FUNCTION F_ROUND_REAL : REAL
VAR_INPUT
  rInput 			: REAL;
  iDecimalPlaces 	: INT;
END_VAR
VAR
  rOutput 			: real;
  rLeftPart 		: REAL;
  Value				: dint;
END_VAR


rOutput := rInput * EXPT(10,iDecimalPlaces);
//rLeftPart := rOutput - TRUNC(rOutput);

//IF rLeftPart >= 0.5 THEN
//  rOutput := rOutput + 1;
//ElSIF rLeftPart <= -0.5 THEN
//  rOutput := rOutput - 1;
//ELSE
//  rOutput := rOutput;
//END_IF

Value := REAL_TO_DINT(rOutput);
rOutput := Value / EXPT(10,iDecimalPlaces);
F_ROUND_REAL := rOutput;

END_FUNCTION

(* stored: Version 1.1.0.1, ProductVersion 3.1.4024.12
   POU F_ROUND_REAL: Id {53dd5f7f-7929-4181-b7a5-b63ad7af92f7}, SpecialFunc None *)
